// vecB = matA * vecA
FUNCTION matMultiVec : bool
VAR_IN_OUT CONSTANT
	matA :ARRAY[*,*] OF LREAL;//m*n
	vecA:ARRAY[*] OF LREAL; // n*1
END_VAR
VAR_IN_OUT 
		vecB :ARRAY[*] OF LREAL;
END_VAR
VAR
	m,n :DINT;
	i,j, k :DINT;
 
END_VAR

m:=UPPER_BOUND(matA,1);
n:= UPPER_BOUND(matA,2);
ASSERT(UPPER_BOUND(vecA,1)=n);
ASSERT(UPPER_BOUND(vecB,1)=n);
FOR i:=1 TO m DO
	vecB[i]:=0.0;
	FOR j:=1 TO n DO
		vecB[i]:=vecB[i]+matA[i,j]*vecA[j];
	END_FOR
END_FOR

END_FUNCTION

(* stored: Version 1.1.0.1, ProductVersion 3.1.4024.12
   POU matMultiVec: Id {8fa1fc4e-9bb5-44b4-829c-607306747973}, SpecialFunc None *)
